TYPE "A0301_Mach_Ribaltatore_Par"
VERSION : 0.1
// Block: A0301_Mach_Ribaltatore_Par
   STRUCT
      SemiAut_Vel : LReal;
      Aut_Vel : LReal;
      Aut_Acc : LReal;
      Aut_Dec : LReal;
      Pos_0 : LReal;
      Pos_1 : LReal;
      Pos_2 : LReal;
      Pos_3 : LReal;
   END_STRUCT;

END_TYPE
